FUNCTION_BLOCK bfb_sun_classifier
  (* Standard: 61499-2 *)
  (* Version 0.1, 2018-00-07, hpea485, UOA *)
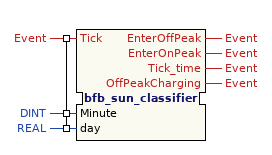
  EVENT_INPUT
    Tick WITH Minute, day;
  END_EVENT
  EVENT_OUTPUT
    EnterOffPeak;
    EnterOnPeak;
    Tick_time;
    OffPeakCharging;
  END_EVENT
  VAR_INPUT
    Minute : DINT;
    day : REAL;
  END_VAR
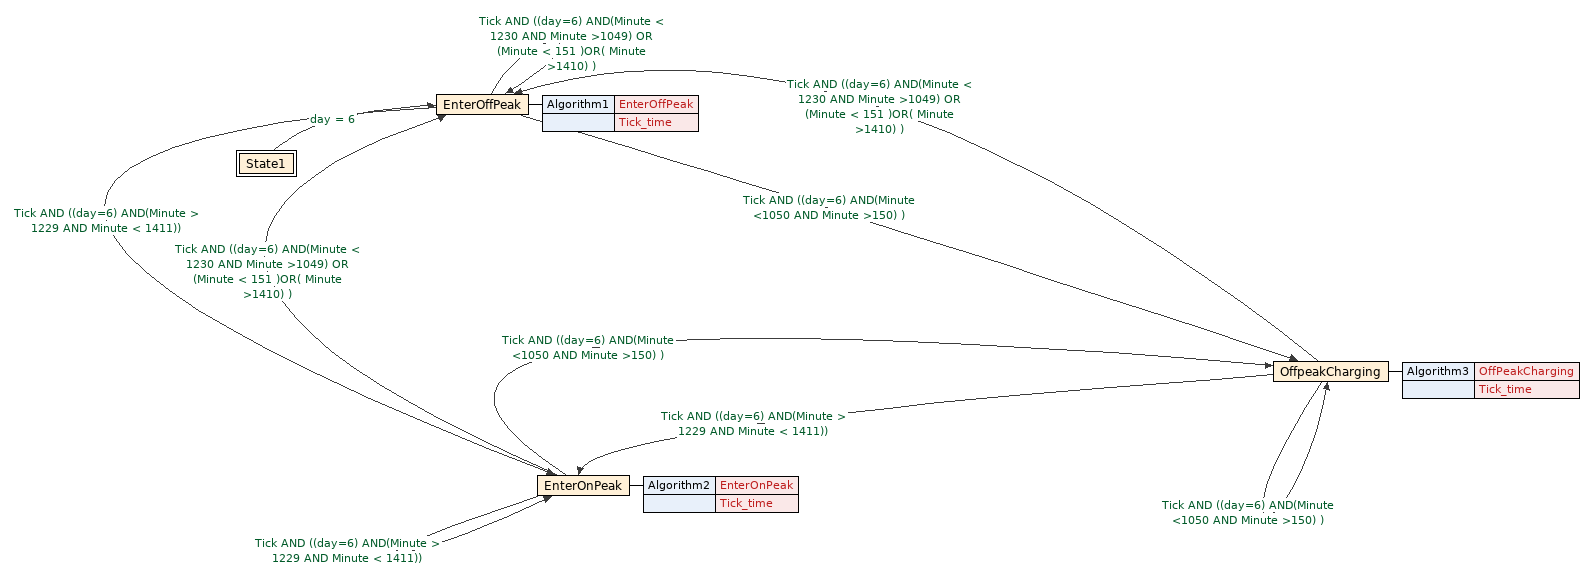
  EC_STATES
    State1;
    EnterOffPeak : Algorithm1 -> EnterOffPeak, -> Tick_time;
    EnterOnPeak : Algorithm2 -> EnterOnPeak, -> Tick_time;
    OffpeakCharging : Algorithm3 -> OffPeakCharging, -> Tick_time;
  END_STATES
  EC_TRANSITIONS
    EnterOffPeak TO EnterOffPeak := Tick AND ((day=6) AND(Minute < 1230 AND Minute >1049) OR (Minute < 151 )OR( Minute >1410) );
    EnterOffPeak TO EnterOnPeak := Tick AND ((day=6) AND(Minute > 1229 AND Minute < 1411));
    EnterOffPeak TO OffpeakCharging := Tick AND ((day=6) AND(Minute <1050 AND Minute >150) );
    EnterOnPeak TO EnterOffPeak := Tick AND ((day=6) AND(Minute < 1230 AND Minute >1049) OR (Minute < 151 )OR( Minute >1410) );
    EnterOnPeak TO EnterOnPeak := Tick AND ((day=6) AND(Minute > 1229 AND Minute < 1411));
    EnterOnPeak TO OffpeakCharging := Tick AND ((day=6) AND(Minute <1050 AND Minute >150) );
    OffpeakCharging TO EnterOnPeak := Tick AND ((day=6) AND(Minute > 1229 AND Minute < 1411));
    OffpeakCharging TO OffpeakCharging := Tick AND ((day=6) AND(Minute <1050 AND Minute >150) );
    OffpeakCharging TO EnterOffPeak := Tick AND ((day=6) AND(Minute < 1230 AND Minute >1049) OR (Minute < 151 )OR( Minute >1410) );
    State1 TO EnterOffPeak := day = 6;
  END_TRANSITIONS
  ALGORITHM Algorithm1 IN C:
printf("Entered OFF PEAK.....\r\n");
  END_ALGORITHM
  ALGORITHM Algorithm2 IN C:
printf(" Entered On peak .....\r\n ");
  END_ALGORITHM
  ALGORITHM Algorithm3 IN C:
printf(" OffPeak Charging \r\n ");
  END_ALGORITHM
END_FUNCTION_BLOCK
